FUNCTION_BLOCK Tieline
  (* Standard: 61499-2 *)
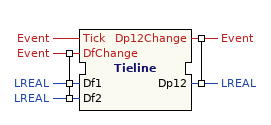
  EVENT_INPUT
    Tick;
    DfChange WITH Df1, Df2;
  END_EVENT
  EVENT_OUTPUT
    Dp12Change WITH Dp12;
  END_EVENT
  VAR_INPUT
    Df1 : LREAL;
    Df2 : LREAL;
  END_VAR
  VAR_OUTPUT
    Dp12 : LREAL;
  END_VAR
  VAR
    StepSize : LREAL := 0.1;
    T0 : LREAL := 0.0707;
    Pi : LREAL := 3.14159;
  END_VAR
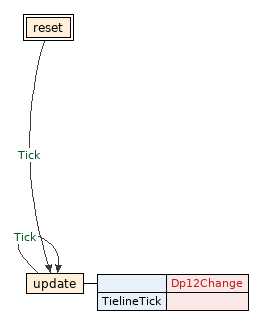
  EC_STATES
    reset;
    update : -> Dp12Change, TielineTick;
  END_STATES
  EC_TRANSITIONS
    reset TO update := Tick;
    update TO update := Tick;
  END_TRANSITIONS
  ALGORITHM TielineTick IN ST:
        Dp12 := Dp12 - (2*Pi*T0*(Df1 - Df2))*StepSize;
  END_ALGORITHM
END_FUNCTION_BLOCK
